// TIA Portal project "Automatic_Sanitization" (V17)
// The Sanitization process should run for 10sec when the door is used 4-times.

(* hardware
DEVICE "S7-1200 station_1"  S7-1200 Station
   slot 0: "Rack_0"  S7-1200 Rack  Rack  V1.0
   slot 1: "PLC_1"  CPU 1212C AC/DC/Rly  6ES7 212-1BE40-0XB0  V4.5
*)

// ===== PLC "PLC_1"  CPU 1212C AC/DC/Rly =====

VAR_GLOBAL   // PLC tag table "Default tag table"
   "unlock_button" AT %I0.0 : Bool;
   "sanitization" AT %Q0.0 : Bool;
   "Tag_1" AT %M0.0 : Bool;
   "Tag_2" AT %M0.1 : Bool;
   "Tag_3" AT %M0.2 : Bool;
   "Tag_4" AT %M0.3 : Bool;
   "Tag_5" AT %M0.4 : Bool;
   "Tag_6" AT %M0.5 : Bool;
   "Tag_7" AT %M0.7 : Bool;
   "Tag_8" AT %M0.6 : Bool;
END_VAR

// folder: System blocks/Program resources

DATA_BLOCK "IEC_Timer_0_DB"   // DB1
{ S7_Optimized_Access := 'TRUE' }
AUTHOR : Simatic
FAMILY : IEC
NAME : IEC_TMR
VERSION : 1.0
// stored: InstanceOfName IEC_TIMER
"IEC_TIMER"
BEGIN
END_DATA_BLOCK

// folder: (top level)

ORGANIZATION_BLOCK "Main"   // OB1, LAD, ProgramCycle
TITLE = "Main Program Sweep (Cycle)"
{ S7_Optimized_Access := 'TRUE' }
VERSION : 0.1
   VAR_INPUT
      Initial_Call : Bool;   // Initial call of this OB
      Remanence : Bool;   // =True, if remanent data are available
   END_VAR
BEGIN

REGION Network 1
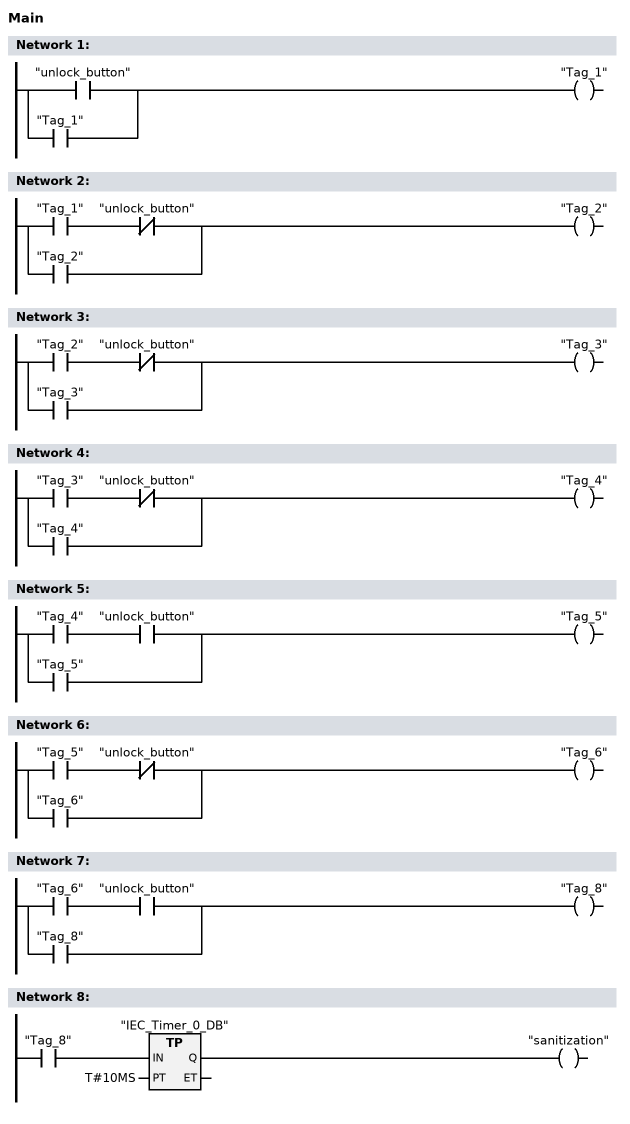
   RUNG wire#powerrail
      Contact( "unlock_button" )
      wire#w1
      Coil( "Tag_1" )
   END_RUNG
   RUNG wire#powerrail
      Contact( "Tag_1" )
   END_RUNG wire#w1
   // the same network as SCL:
   "Tag_1" := "unlock_button" OR "Tag_1";
END_REGION

REGION Network 2
   RUNG wire#powerrail
      Contact( "Tag_1" )
      I_Contact( "unlock_button" )
      wire#w1
      Coil( "Tag_2" )
   END_RUNG
   RUNG wire#powerrail
      Contact( "Tag_2" )
   END_RUNG wire#w1
   // the same network as SCL:
   "Tag_2" := ("Tag_1" AND NOT "unlock_button") OR "Tag_2";
END_REGION

REGION Network 3
   RUNG wire#powerrail
      Contact( "Tag_2" )
      I_Contact( "unlock_button" )
      wire#w1
      Coil( "Tag_3" )
   END_RUNG
   RUNG wire#powerrail
      Contact( "Tag_3" )
   END_RUNG wire#w1
   // the same network as SCL:
   "Tag_3" := ("Tag_2" AND NOT "unlock_button") OR "Tag_3";
END_REGION

REGION Network 4
   RUNG wire#powerrail
      Contact( "Tag_3" )
      I_Contact( "unlock_button" )
      wire#w1
      Coil( "Tag_4" )
   END_RUNG
   RUNG wire#powerrail
      Contact( "Tag_4" )
   END_RUNG wire#w1
   // the same network as SCL:
   "Tag_4" := ("Tag_3" AND NOT "unlock_button") OR "Tag_4";
END_REGION

REGION Network 5
   RUNG wire#powerrail
      Contact( "Tag_4" )
      Contact( "unlock_button" )
      wire#w1
      Coil( "Tag_5" )
   END_RUNG
   RUNG wire#powerrail
      Contact( "Tag_5" )
   END_RUNG wire#w1
   // the same network as SCL:
   "Tag_5" := ("Tag_4" AND "unlock_button") OR "Tag_5";
END_REGION

REGION Network 6
   RUNG wire#powerrail
      Contact( "Tag_5" )
      I_Contact( "unlock_button" )
      wire#w1
      Coil( "Tag_6" )
   END_RUNG
   RUNG wire#powerrail
      Contact( "Tag_6" )
   END_RUNG wire#w1
   // the same network as SCL:
   "Tag_6" := ("Tag_5" AND NOT "unlock_button") OR "Tag_6";
END_REGION

REGION Network 7
   RUNG wire#powerrail
      Contact( "Tag_6" )
      Contact( "unlock_button" )
      wire#w1
      Coil( "Tag_8" )
   END_RUNG
   RUNG wire#powerrail
      Contact( "Tag_8" )
   END_RUNG wire#w1
   // the same network as SCL:
   "Tag_8" := ("Tag_6" AND "unlock_button") OR "Tag_8";
END_REGION

REGION Network 8
   "IEC_Timer_0_DB".TP(IN := "Tag_8", PT := T#10MS);
   "sanitization" := "IEC_Timer_0_DB".Q;
END_REGION
END_ORGANIZATION_BLOCK